// TwinCAT 3 PLC project Oefeningen1
// ProgramVersion: 3.1.4026.18
// libraries:
//   Tc2_BABasic, * (Beckhoff Automation GmbH)
//   Tc2_Standard, * (Beckhoff Automation GmbH)
//   Tc2_System, * (Beckhoff Automation GmbH)
//   Tc3_Module, * (Beckhoff Automation GmbH)
// project tree:
//   / GlobalTextList.TcGTLO, PlcTask.TcTTO, Visualization Manager.TcVMO (not stored)
//   POUs/ MAIN.TcPOU, prg_Alarmbewaking.TcPOU, prg_DriePompen.TcPOU, prg_Verschalingmetfunctie.TcPOU, prg_jafunctie.TcPOU, prg_MotorMetDrukknop.TcPOU, PRG_OpslagFoutDetectie.TcPOU, prg_Opslagvat.TcPOU, prg_Reactorvat.TcPOU, prg_Teleruptorschakeling.TcPOU, prg_TweePompen.TcPOU, prg_TweeSignalen.TcPOU
//   VISUs/ Visualization_MotorMetDrukknop.TcVIS
// real-time tasks:
//   TASK PlcTask: cycle T#10ms, priority 20, ADS port 350
//   TASK PlcTask1: cycle T#10ms, priority 21, ADS port 351
//   TASK PlcTask2: cycle T#10ms, priority 22, ADS port 352
//   TASK PlcTask3: cycle T#10ms, priority 23, ADS port 353
//   TASK PlcTask4: cycle T#10ms, priority 24, ADS port 354

CONFIGURATION Oefeningen1
    RESOURCE PLC ON TwinCAT3
        TASK PlcTask(INTERVAL := T#10ms, PRIORITY := 20);
        PROGRAM MAIN WITH PlcTask : MAIN;
    END_RESOURCE
END_CONFIGURATION

// ---- POUs/MAIN.TcPOU
PROGRAM MAIN
VAR
END_VAR

//prg_jafunctie();
//prg_TweeSignalen();
//prg_Reactorvat();
//prg_Opslagvat();
//PRG_OpslagFoutDetectie();
//prg_Alarmbewaking();
//prg_Teleruptorschakeling();
//prg_MotorMetDrukknop();
//prg_TweePompen();
//prg_DriePompen();
prg_Verschalingmetfunctie();

END_PROGRAM

// ---- POUs/prg_Verschalingmetfunctie.TcPOU
PROGRAM prg_Verschalingmetfunctie
VAR
	//POTENTIOMETERRRR
	//0 tot 32767
	nPotentiometer		AT		%I*		:INT;
	nPotentiometerValue		:INT;
	nPower				AT		%Q*		:INT:=32767;
	
	//DISPLAYYYYY
	//–100 tot +2 000
	nDisplay			AT		%Q*		:INT;
END_VAR


//Hier wordt de data van potentiometer van 0 tot 30 verschaald
nPotentiometer:=TO_INT(F_Scale(
	fRawData:= nPotentiometerValue, 
	fRawDataLowerOffLimit:= 0, 
	fRawDataUpperOffLimit:= 32767, 
	fScaleDataLowerOffLimit:= 0, 
	fScaleDataUpperOffLimit:= 10));
	
	
//DUS NU WORDT DE DATA VAN nDisplay van 0 tot 1000 verschaald
nDisplay:=TO_INT(F_Scale(
	fRawData:= nPotentiometer, 
	fRawDataLowerOffLimit:= 0, 
	fRawDataUpperOffLimit:= 10, 
	fScaleDataLowerOffLimit:= 0, 
	fScaleDataUpperOffLimit:= 1000));

END_PROGRAM

// ---- POUs/prg_Alarmbewaking.TcPOU
PROGRAM prg_Alarmbewaking
VAR
	Sensor1		AT		%I*		:BOOL; //Druk Te Hoog (True)
	Sensor2		AT		%I*		:BOOL; //Temperatuur Te Hoog (True)
	Sensor3		AT		%I*		:BOOL; //Laag vloeistof (True) In de oefening moet dit false zijn maar dit is gewoon verwarrend maak er dan NOT(..) van waar deze voorkomt in het programma
	DrukKnop	AT		%I*		:BOOL;
	
	Lamp1		AT		%Q*		:BOOL; //Druk Te Hoog
	Lamp2		AT		%Q*		:BOOL; //Temperatuur Te Hoog
	Lamp3		AT		%Q*		:BOOL; //Vloeistof Te Laag
	Lamp4		AT		%Q*		:BOOL; //TweeAlarmen
	Lamp5		AT		%Q*		:BOOL; //Drie Alarmen
	
	
	SetReset: SR;
END_VAR

Lamp1 := Sensor1;
Lamp2 := Sensor2;
Lamp3 := Sensor3;

Lamp4 := (NOT(Sensor1) AND Sensor2 AND Sensor3) OR
		 (Sensor1 AND NOT(Sensor2) AND Sensor3) OR
		 (Sensor1 AND Sensor2 AND NOT Sensor3);

SetReset(SET1:= Sensor1 AND Sensor2 AND Sensor3, RESET:=DrukKnop , Q1=> Lamp5);

END_PROGRAM

// ---- POUs/prg_DriePompen.TcPOU
PROGRAM prg_DriePompen
VAR
	Hoofdschakelaar		AT		%I*		:BOOL;
	Drukknop			AT		%I*		:BOOL;
	StopKnop			AT		%I*		:BOOL;
	
	Pomp1				AT		%Q*		:BOOL;
	Pomp2				AT		%Q*		:BOOL;
	Pomp3				AT		%Q*		:BOOL;
	DrukOpKnop: R_TRIG;
END_VAR

IF Hoofdschakelaar AND NOT StopKnop THEN
	DrukOpKnop(CLK:= Drukknop);
ELSE	
	Pomp1:=FALSE;
	Pomp2:=FALSE;
	Pomp3:=FALSE;
END_IF
IF DrukOpKnop.Q AND NOT Pomp1 AND NOT Pomp2 AND NOT Pomp3 THEN
	Pomp1:=TRUE;
ELSIF DrukOpKnop.Q AND Pomp1 AND NOT Pomp2 AND NOT Pomp3 THEN
	Pomp1:=TRUE;
	Pomp2:=TRUE;
ELSIF DrukOpKnop.Q AND  Pomp1 AND Pomp2 AND NOT Pomp3 THEN
	Pomp1:=TRUE;
	Pomp2:=TRUE;
	Pomp3:=TRUE;
ELSIF DrukOpKnop.Q AND  Pomp1 AND Pomp2 AND Pomp3 THEN
	Pomp1:=FALSE;
	Pomp2:=FALSE;
	Pomp3:=FALSE;
END_IF

END_PROGRAM

// ---- POUs/prg_jafunctie.TcPOU
PROGRAM prg_jafunctie
VAR
	Ingang		AT		%I*		:BOOL;
	Uitgang		AT		%Q*		:BOOL;
END_VAR

Uitgang := Ingang;

END_PROGRAM

// ---- POUs/prg_MotorMetDrukknop.TcPOU
PROGRAM prg_MotorMetDrukknop
VAR
  	T1: R_TRIG;
	Drukknop		AT		%I*		:BOOL;
	Hoofdschakelaar	AT		%I*		:BOOL;
	
	MotorLinks		AT		%Q*		:BOOL;
	MotorRechts		AT		%Q*		:BOOL;

	Switch: BOOL;
END_VAR

T1(CLK := Drukknop);

IF Hoofdschakelaar AND T1.Q THEN
    IF MotorLinks OR MotorRechts THEN
        MotorLinks := FALSE;
        MotorRechts := FALSE;
        Switch := NOT Switch;
    ELSIF NOT Switch THEN
        MotorLinks := TRUE;
    ELSE
        MotorRechts := TRUE;
    END_IF
END_IF

END_PROGRAM

// ---- POUs/PRG_OpslagFoutDetectie.TcPOU
PROGRAM PRG_OpslagFoutDetectie
VAR
	SensorHoog		AT		%I*		:BOOL;
	SensorLaag		AT		%I*		:BOOL;
	StartKnop		AT		%I*		:BOOL;
	StopKnop		AT		%I*		:BOOL;
	
	Klep			AT		%Q*		:BOOL;
	Pomp			AT		%Q*		:BOOL;
	Vullen			AT		%Q*		:BOOL;
END_VAR

Klep := SensorLaag AND NOT(SensorHoog);
Vullen := SensorLaag AND NOT(SensorHoog);

IF StopKnop OR Vullen OR NOT(SensorLaag) OR (SensorLaag AND NOT(SensorHoog)) OR NOT(StartKnop) THEN
	Pomp := FALSE;
ELSIF StartKnop THEN
	Pomp := TRUE; 
END_IF

END_PROGRAM

// ---- POUs/prg_Opslagvat.TcPOU
PROGRAM prg_Opslagvat
VAR
	SensorHoog		AT		%I*		:BOOL;
	SensorLaag		AT		%I*		:BOOL;
	StartKnop		AT		%I*		:BOOL;
	StopKnop		AT		%I*		:BOOL;
	
	Klep			AT		%Q*		:BOOL;
	Pomp			AT		%Q*		:BOOL;
	Vullen			AT		%Q*		:BOOL;
END_VAR

Klep := SensorLaag AND NOT(SensorHoog);
Vullen := SensorLaag AND NOT(SensorHoog);

IF StopKnop OR Vullen OR (SensorLaag AND NOT(SensorHoog)) THEN
	Pomp := FALSE;
ELSIF StartKnop THEN
	Pomp := TRUE; 
END_IF

END_PROGRAM

// ---- POUs/prg_Reactorvat.TcPOU
PROGRAM prg_Reactorvat
VAR
	S01			AT		%I*		:BOOL;	//NiveauTeHoog
	S02			AT		%I*		:BOOL;	//TemperatuurTeHoog
	S03			AT		%I*		:BOOL;  //DrukTeHoog
	S04			AT		%I*		:BOOL;	//StopKnop Normaal Gesloten
	S05			AT		%I*		:BOOL;	//HoofdSchakelaar
	
	Q01			AT		%Q*		:BOOL;	//OranjeLamp (bij detectie 1 sensor)
	Q02			AT		%Q*		:BOOL;	//RodeLamp (bij detectie 2 sensor)
	Q05			AT		%Q*		:BOOL;	//AlarmBel (bij detectie 3 sensor)
END_VAR

Q01 := S05 AND (S01 OR S02 OR S03);
Q02 := S05 AND ((S01 AND S02) OR
			    (S01 AND S03) OR
			    (S02 AND S03));
Q05 := (NOT(S04) AND S05) AND (S01 AND S02 AND S03);

END_PROGRAM

// ---- POUs/prg_Teleruptorschakeling.TcPOU
PROGRAM prg_Teleruptorschakeling
VAR
	Drukknop1		AT		%I*		:BOOL;
	Drukknop2		AT		%I*		:BOOL;
	Drukknop3		AT		%I*		:BOOL;
	
	Verlichting		AT		%Q*		:BOOL;
	RisingEdge: R_TRIG;
END_VAR

RisingEdge(CLK := Drukknop1 OR Drukknop2 OR Drukknop3);

IF RisingEdge.Q THEN
    Verlichting := NOT Verlichting; //Wisselt tussen Aan en uit, als hij aan is wordt hij NOT aan dus uit, als hij uit is wordt hij NOT uit dus aan
END_IF

END_PROGRAM

// ---- POUs/prg_TweePompen.TcPOU
PROGRAM prg_TweePompen
VAR
	Hoofdschakelaar			AT		%I*		:BOOL;
	StartKnop				AT		%I*		:BOOL;
	StopKnop				AT		%I*		:BOOL;
	NiveauSchakelaarOnder	AT		%I*		:BOOL;
	NiveauSchakelaarBoven	AT		%I*		:BOOL;
	
	Pomp1					AT		%Q*		:BOOL;
	Pomp2					AT		%Q*		:BOOL;
	PompWissel: BOOL;
	PompAan: BOOL;
	
END_VAR

IF Hoofdschakelaar AND (StartKnop OR NiveauSchakelaarOnder) AND NOT (StopKnop OR NiveauSchakelaarBoven) THEN
	PompAan:=TRUE;
ELSE
	PompAan:=False;	
END_IF

IF PompAan AND NOT Pomp1 AND NOT Pomp2 THEN
	PompWissel:= NOT PompWissel;
END_IF

IF PompAan THEN
    Pomp1 := PompWissel;
    Pomp2 := NOT PompWissel;
ELSE
    Pomp1 := FALSE;
    Pomp2 := FALSE;
END_IF

END_PROGRAM

// ---- POUs/prg_TweeSignalen.TcPOU
PROGRAM prg_TweeSignalen
VAR
	S01, S02		AT		%I*		:BOOL; 
	Q01, Q02		AT		%Q*		:BOOL;
END_VAR

Q01 := NOT(S02);
Q02 := NOT(S01);

END_PROGRAM

// ---- GlobalTextList.TcGTLO
TEXTLIST GlobalTextList
  430 = 'Drukknop'
  951 = 'MotorLinks'
  960 = 'MotorRechts'
END_TEXTLIST

// ---- VISUs/Visualization_MotorMetDrukknop.TcVIS
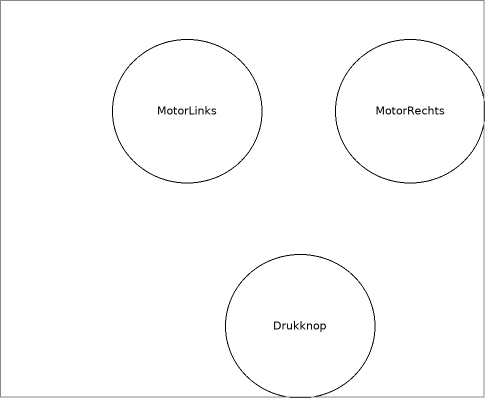
VISUALIZATION Visualization_MotorMetDrukknop  // 485x398
    Ellipse (112,39 150x144), "MotorLinks", colour toggle: prg_MotorMetDrukknop.MotorLinks
    Ellipse (225,254 150x144), "Drukknop"
        tap prg_MotorMetDrukknop.Drukknop
    Ellipse (335,39 150x144), "MotorRechts", colour toggle: prg_MotorMetDrukknop.MotorRechts
END_VISUALIZATION
